{attribute 'qualified_only'}
VAR_GLOBAL
	stMainProcess		: ST_StageProcess;
END_VAR

(* stored: Version 1.1.0.1, ProductVersion 3.1.4024.11
   GVL GVL_Main: Id {a79c6a64-f573-4368-841c-eec0feaaebf4} *)
